FUNCTION_BLOCK FB_HeartbeatDetect
VAR_INPUT
END_VAR
VAR_OUTPUT
END_VAR
VAR
	m_heartbeatLowCount :INT :=0;
	m_heartbeatHighCount :INT :=0;
	m_heartbeatCountThres :INT :=500;
END_VAR

// check if instrument is on
METHOD run : BOOL
VAR_INPUT
	IOValue :UDINT;
END_VAR
//heartbeat cycle 100ms
IF IOValue = 0 THEN
	m_heartbeatHighCount:=0;
	m_heartbeatLowCount :=MIN(m_heartbeatLowCount +1,2*m_heartbeatCountThres);
ELSIF  IOValue = 1 THEN
	m_heartbeatLowCount:=0;
	m_heartbeatHighCount :=MIN(m_heartbeatHighCount +1,2*m_heartbeatCountThres);
END_IF

run := NOT(m_heartbeatLowCount >= m_heartbeatCountThres OR m_heartbeatHighCount>=m_heartbeatCountThres);
END_METHOD

END_FUNCTION_BLOCK

(* stored: Version 1.1.0.1, ProductVersion 3.1.4024.11
   POU FB_HeartbeatDetect: Id {486f1896-2368-4412-bcb6-b0e058b4d35b}, SpecialFunc None
   Method run: Id {3e7a4fc3-a1b0-4ce0-ad1f-146139077201} *)
